FUNCTION_BLOCK FB_TsFBEDM_Diag
VAR_INPUT
	nDiag		: USINT;
END_VAR
VAR_OUTPUT
	sDiag		: STRING;
END_VAR
VAR
END_VAR

CASE nDiag OF
	0:		sDiag := 'No Error';		
	1:		sDiag := 'Switch-OFF timer elapsed';	
	2:		sDiag := 'Switch-ON timer elapsed';	
ELSE 
	sDiag := 'undefined';
END_CASE

END_FUNCTION_BLOCK

(* stored: Version 1.1.0.1, ProductVersion 3.1.4024.15
   POU FB_TsFBEDM_Diag: Id {36e2d0bb-907a-4162-ab81-bea962fcf5fc}, SpecialFunc None *)
